(* CODESYS project SmartConveyorVirtualCommissioning.project

Project tree, tasks and I/O mapping:
  Device : CODESYS Control Win V3 x64, CODESYS, version 3.5.22.30
    application Application
      libraries: Standard, 3.5.22.0 (System)
      task MainTask (cyclic, interval t#20ms, priority 1) calls PLC_PRG
      var PLC_PRG [ST]
      global variables FIO
      Symbols
      data type E_SequenceState
      data type E_OperatingMode
*)

// Device/Application/E_SequenceState
{attribute 'qualified_only'}
{attribute 'strict'}
TYPE E_SequenceState :
(
    SEQ_IDLE := 0,
    SEQ_LOADING := 10,
    SEQ_ROTATE_TO_UNLOAD := 20,
    SEQ_DISCHARGING := 30,
    SEQ_RETURN_TO_LOAD := 40
);
END_TYPE

// Device/Application/E_OperatingMode
{attribute 'qualified_only'}
{attribute 'strict'}
TYPE E_OperatingMode :
(
    MODE_OFF := 0,
    MODE_MANUAL := 10,
    MODE_AUTO := 20
);
END_TYPE

// Device/Application/FIO
{attribute 'qualified_only'}
VAR_GLOBAL
    iAtEntry 		: BOOL;
    iLowBox 		: BOOL;
    iHighBox 		: BOOL;
    iAtTurnEntry 	: BOOL;
    iAtLoadPos		: BOOL;
    iAtUnloadPos 	: BOOL;
    iAtFront		: BOOL;
    iAtRightEntry	: BOOL;
    iAtLeftEntry	: BOOL;
    iAtRightExit	: BOOL;
    iAtLeftExit		: BOOL;
 
    oFeederConveyor	: BOOL;
    oEntryConveyor 	: BOOL;
    oLoad			: BOOL;
    oUnload			: BOOL;
    oTurn			: BOOL;
    oLeftConveyor	: BOOL;
    oRightConveyor	: BOOL;
END_VAR

// Device/Application/PLC_PRG
VAR
    (* Edge detection *)
    F_AtEntry       : F_TRIG;
    F_AtTurnEntry   : F_TRIG;
    F_AtRightEntry  : F_TRIG;
    F_AtLeftEntry   : F_TRIG;
    F_AtRightExit   : F_TRIG;
    F_AtLeftExit    : F_TRIG;


    (* Feedback *)
    xAtEntry        : BOOL;
    xAtFront        : BOOL;
    xAtLeftEntry    : BOOL;
    xAtLeftExit     : BOOL;
    xAtLoadPos      : BOOL;
    xAtRightEntry   : BOOL;
    xAtRightExit    : BOOL;
    xAtTurnEntry    : BOOL;
    xAtUnloadPos    : BOOL;
    xHighBox        : BOOL;
    xLowBox         : BOOL;


    (* Operating mode *)
    eOperatingMode  : E_OperatingMode := E_OperatingMode.MODE_OFF;


    (* Operator requests - behaviour added in Week 2 *)
    xOpStart        : BOOL;
    xOpStop         : BOOL;
    xOpReset        : BOOL;


    (* Sequence *)
    eSequenceState  : E_SequenceState := E_SequenceState.SEQ_IDLE;


    (* Machine status *)
    xReady          : BOOL;
    xRunning        : BOOL;


    (* Machine internal state - existing sample behaviour *)
    Pallet_on_left      : BOOL := FALSE;
    Pallet_on_right     : BOOL := FALSE;
    Turntable_busy      : BOOL := FALSE;
    Discharge_direction : BOOL := FALSE;
    Entry_busy          : BOOL := FALSE;
    Pallet_on_entry     : BOOL := FALSE;
    Count               : WORD := 16#8000;


    (* Permissives - logic added later *)
    xPermissiveRun       : BOOL;
    xPermissiveRotation  : BOOL;
    xPermissiveDischarge : BOOL;


    (* Fault framework - implementation added later *)
    xFaultActive    : BOOL;


    (* Actuator commands *)
    xCmdEntryConveyor  : BOOL;
    xCmdFeederConveyor : BOOL;
    xCmdLeftConveyor   : BOOL;
    xCmdLoad           : BOOL;
    xCmdRightConveyor  : BOOL;
    xCmdTurn           : BOOL;
    xCmdUnload         : BOOL;
END_VAR

(**** INPUT MAPPING ****)
xAtEntry       := FIO.iAtEntry;
xAtFront       := FIO.iAtFront;
xAtLeftEntry   := FIO.iAtLeftEntry;
xAtLeftExit    := FIO.iAtLeftExit;
xAtLoadPos     := FIO.iAtLoadPos;
xAtRightEntry  := FIO.iAtRightEntry;
xAtRightExit   := FIO.iAtRightExit;
xAtTurnEntry   := FIO.iAtTurnEntry;
xAtUnloadPos   := FIO.iAtUnloadPos;
xHighBox       := FIO.iHighBox;
xLowBox        := FIO.iLowBox;

F_AtEntry(CLK := xAtEntry);
F_AtTurnEntry(CLK := xAtTurnEntry);
F_AtRightEntry(CLK := xAtRightEntry);	           
F_AtLeftEntry(CLK := xAtLeftEntry);		(* A pallet abandons the turntable, being charged onto the left exit conveyer *)
F_AtRightExit(CLK := xAtRightExit);
F_AtLeftExit(CLK := xAtLeftExit); 		(* A pallet abandons the left exit conveyer *)

(**** LEFT EXIT CONVEYER CONTROL ****)
(* Pallet_on_left represents the state of the left exit conveyer: if it carries a pallet, then Pallet_on_left = TRUE *)

IF F_AtLeftExit.Q THEN						(* When a pallet abandons the conveyer *)
	Pallet_on_left := FALSE;				(* Reset Pallet_on_left *)
END_IF;

IF xAtLeftEntry THEN 					(* When there’s a pallet at the entry of the conveyer *)
	Pallet_on_left := TRUE;					(* Set Pallet_on_left *)
END_IF;

xCmdLeftConveyor := Pallet_on_left;		(* Left exit conveyer runs for Pallet_on_left = TRUE *)

(**** RIGHT EXIT CONVEYER CONTROL ****)
IF F_AtRightExit.Q THEN  	
	Pallet_on_right := FALSE;
END_IF;

IF xAtRightEntry THEN		
	Pallet_on_right := TRUE;	
END_IF;

xCmdRightConveyor := Pallet_on_right;

(**** TURNTABLE SEQUENCE ****)
CASE eSequenceState OF

    E_SequenceState.SEQ_IDLE:
        IF xAtTurnEntry THEN
            eSequenceState := E_SequenceState.SEQ_LOADING;
        END_IF;

    E_SequenceState.SEQ_LOADING:
        IF xAtFront THEN
            eSequenceState := E_SequenceState.SEQ_ROTATE_TO_UNLOAD;
        END_IF;

    E_SequenceState.SEQ_ROTATE_TO_UNLOAD:
        IF xAtUnloadPos THEN
            eSequenceState := E_SequenceState.SEQ_DISCHARGING;
        END_IF;

    E_SequenceState.SEQ_DISCHARGING:
        IF F_AtRightEntry.Q OR F_AtLeftEntry.Q THEN
            eSequenceState := E_SequenceState.SEQ_RETURN_TO_LOAD;
        END_IF;

    E_SequenceState.SEQ_RETURN_TO_LOAD:
        IF xAtLoadPos THEN
            eSequenceState := E_SequenceState.SEQ_IDLE;
        END_IF;

ELSE
    eSequenceState := E_SequenceState.SEQ_IDLE;

END_CASE;

IF F_AtTurnEntry.Q THEN
    Turntable_busy := TRUE;
END_IF;

IF eSequenceState = E_SequenceState.SEQ_IDLE THEN
    Turntable_busy := FALSE;
END_IF;

xCmdLoad :=
    (eSequenceState = E_SequenceState.SEQ_LOADING)
    OR
    ((eSequenceState = E_SequenceState.SEQ_DISCHARGING)
    AND Discharge_direction);

xCmdUnload :=
    (eSequenceState = E_SequenceState.SEQ_DISCHARGING)
    AND NOT Discharge_direction;

xCmdTurn :=
    (eSequenceState = E_SequenceState.SEQ_ROTATE_TO_UNLOAD)
    OR
    (eSequenceState = E_SequenceState.SEQ_DISCHARGING);

(**** ENTRY CONVEYER CONTROL ****)

IF F_AtEntry.Q THEN 			
	Count := ROL (Count,1);		
	IF (Count = WORD#16#2) THEN	
		Entry_busy := TRUE; 			
	END_IF;	
END_IF;

IF F_AtTurnEntry.Q THEN  			
	Discharge_direction := NOT Discharge_direction;

	(** Defining the direction of the discharge: the direction of the discharge changes every time a pallet is discharged from the entry conveyer onto the turntable. If Discharge_direction = FALSE, then the discharge is onto the right conveyer **)

	Entry_busy := FALSE;	 		
	Count := ROR(Count,1); 	
	IF (Count = WORD#16#8000) THEN	
		Pallet_on_entry := FALSE; 			
	END_IF;
END_IF;

IF xAtEntry THEN		
	Pallet_on_entry := TRUE;	 	
END_IF;
				
xCmdEntryConveyor :=
    Pallet_on_entry AND
    (NOT Turntable_busy OR NOT xAtTurnEntry);

(**** FEEDING CONVEYER CONTROL ****)
xCmdFeederConveyor :=
    NOT Entry_busy OR NOT xAtEntry;

(**** OUTPUT MAPPING ****)
FIO.oEntryConveyor  := xCmdEntryConveyor;
FIO.oFeederConveyor := xCmdFeederConveyor;
FIO.oLeftConveyor   := xCmdLeftConveyor;
FIO.oLoad           := xCmdLoad;
FIO.oRightConveyor  := xCmdRightConveyor;
FIO.oTurn           := xCmdTurn;
FIO.oUnload         := xCmdUnload;
